(*
    Control module for one discrete sensor point: the leaf every miniload
    equipment module reads its world through.

    Three stages, in this order, and the order is the contract:

      1. source select - SimulatedInput replaces HardwareInput while Simulation
         is set, so a mock feeds the SAME filter the field bit does;
      2. polarity     - Inverted negates the selected level, so a normally
         closed device debounces on what the signal MEANS;
      3. debounce     - a symmetric on-delay/off-delay pair. Active may only
         rise once the level has held high for DebounceTime, and may only fall
         once it has held low for DebounceTime. Between those two windows
         Active holds its previous value, which is what makes a chattering
         photo-eye a no-op instead of a burst of transitions.

    TimeActive and TimeInactive meter the settled state, not the wire, and each
    resets when Active moves. A conveyor asks TimeInactive "has the lane been
    clear long enough to hand over"; a diagnostic asks TimeActive "has this
    photo-eye been blocked too long".
*)
FUNCTION_BLOCK FB_DigitalInput IMPLEMENTS I_DigitalInput
VAR_INPUT
	// The field bit, wired to a terminal channel on a real machine.
	HardwareInput : BOOL;
END_VAR
VAR_OUTPUT
	Data : ST_SensorData;
END_VAR
VAR
	sourceLevel : BOOL;
	signalLevel : BOOL;
	settled : BOOL;
	invert : BOOL;
	simulate : BOOL;
	simulatedLevel : BOOL;
	debounce : TIME;
	riseFilter : TON;
	fallFilter : TOF;
	activeMeter : TON;
	inactiveMeter : TON;
	// The elapsed meters are on-delays that are never meant to fire: their PT
	// only has to outlast any stretch worth measuring, because ET is capped at
	// PT. Well inside TIME's 49-day range, so no wrap.
	MeterCeiling : TIME := T#24d;
END_VAR

// Source select
IF simulate THEN
	sourceLevel := simulatedLevel;
ELSE
	sourceLevel := HardwareInput;
END_IF

// Polarity
signalLevel := sourceLevel XOR invert;

// Debounce. riseFilter.Q means "high, continuously, for at least DebounceTime";
// fallFilter.Q stays TRUE until the level has been low that same span, so
// NOT fallFilter.Q is its mirror. Neither true means the level is still inside
// a settling window and the last settled value stands.
riseFilter(IN := signalLevel, PT := debounce);
fallFilter(IN := signalLevel, PT := debounce);

IF riseFilter.Q THEN
	settled := TRUE;
ELSIF NOT fallFilter.Q THEN
	settled := FALSE;
END_IF

// Elapsed meters. Driven by the settled state rather than signalLevel, so a
// bounce that never reached Active never disturbs them either.
activeMeter(IN := settled, PT := MeterCeiling);
inactiveMeter(IN := NOT settled, PT := MeterCeiling);

// Status
Data.Active := settled;
Data.RawLevel := sourceLevel;
Data.Inverted := invert;
Data.Simulated := simulate;
Data.DebounceTime := debounce;
Data.TimeActive := activeMeter.ET;
Data.TimeInactive := inactiveMeter.ET;

PROPERTY Active : BOOL
GET
Active := settled;
END_GET
END_PROPERTY

PROPERTY DebounceTime : TIME
GET
DebounceTime := debounce;
END_GET
SET
debounce := DebounceTime;
END_SET
END_PROPERTY

PROPERTY Inverted : BOOL
GET
Inverted := invert;
END_GET
SET
invert := Inverted;
END_SET
END_PROPERTY

PROPERTY Simulation : BOOL
GET
Simulation := simulate;
END_GET
SET
simulate := Simulation;
END_SET
END_PROPERTY

PROPERTY SimulatedInput : BOOL
GET
SimulatedInput := simulatedLevel;
END_GET
SET
simulatedLevel := SimulatedInput;
END_SET
END_PROPERTY

PROPERTY TimeActive : TIME
GET
TimeActive := activeMeter.ET;
END_GET
END_PROPERTY

PROPERTY TimeInactive : TIME
GET
TimeInactive := inactiveMeter.ET;
END_GET
END_PROPERTY

END_FUNCTION_BLOCK

(* stored: Version 1.1.0.1, ProductVersion 3.1.4026.18
   POU FB_DigitalInput: Id {5e4501d0-0003-4d19-9a41-000000000001}, SpecialFunc None
   Property Active: Id {5e4501d0-0003-4d19-9a41-000000000002}
   Get Get: Id {5e4501d0-0003-4d19-9a41-000000000003}
   Property DebounceTime: Id {5e4501d0-0003-4d19-9a41-000000000004}
   Get Get: Id {5e4501d0-0003-4d19-9a41-000000000005}
   Set Set: Id {5e4501d0-0003-4d19-9a41-000000000006}
   Property Inverted: Id {5e4501d0-0003-4d19-9a41-000000000007}
   Get Get: Id {5e4501d0-0003-4d19-9a41-000000000008}
   Set Set: Id {5e4501d0-0003-4d19-9a41-000000000009}
   Property Simulation: Id {5e4501d0-0003-4d19-9a41-00000000000a}
   Get Get: Id {5e4501d0-0003-4d19-9a41-00000000000b}
   Set Set: Id {5e4501d0-0003-4d19-9a41-00000000000c}
   Property SimulatedInput: Id {5e4501d0-0003-4d19-9a41-00000000000d}
   Get Get: Id {5e4501d0-0003-4d19-9a41-00000000000e}
   Set Set: Id {5e4501d0-0003-4d19-9a41-00000000000f}
   Property TimeActive: Id {5e4501d0-0003-4d19-9a41-000000000010}
   Get Get: Id {5e4501d0-0003-4d19-9a41-000000000011}
   Property TimeInactive: Id {5e4501d0-0003-4d19-9a41-000000000012}
   Get Get: Id {5e4501d0-0003-4d19-9a41-000000000013} *)
